// TIA Portal V17 export
// export: Created 2022-07-20T06:59:50.0989637Z, ExportSetting WithDefaults, DisplayName Totally Integrated Automation Portal, DisplayVersion V17, DisplayName TIA Portal Openness, DisplayVersion V17, DisplayName TIA Portal Version Control Interface, DisplayVersion V17, DisplayName SINAMICS Startdrive Advanced, DisplayVersion V17, DisplayName SINAMICS Startdrive G130, G150, S120, S150, SINAMICS MV, S210, DisplayVersion V17, DisplayName SINAMICS Startdrive G110M, G120, G120C, G120D, G120P, G115D, DisplayVersion V17, DisplayName STEP 7 Professional, DisplayVersion V17, DisplayName STEP 7 Safety, DisplayVersion V17, DisplayName WinCC Advanced, DisplayVersion V17
FUNCTION_BLOCK "FB10022_Average"   // FB10022, LAD
{ S7_Optimized_Access := 'TRUE' }
VERSION : 0.1
// stored: AutoNumber false, IsIECCheckEnabled false, IsRetainMemResEnabled false, MemoryReserve 100, SetENOAutomatically false, UDAEnableTagReadback false
   VAR_INPUT
      Value : Real;
      Clock : Bool;
      Clear : Bool;
   END_VAR
   VAR_OUTPUT
      Result : Real;
   END_VAR
   VAR_IN_OUT
      Items : Array[*] of Real;
   END_VAR
   VAR
      R_TRIG_Clock : R_TRIG;
      statItemNumber { S7_SetPoint := 'True'} : DInt;
      statStartElement : DInt;
      statEndElement : DInt;
      statItemsFull : Bool;
   END_VAR
   VAR_TEMP
      iItem : Int;
   END_VAR
BEGIN

REGION Network 1 (SCL): First Scan
   IF "FirstScan" THEN
       #statStartElement := LOWER_BOUND(ARR := #Items, DIM := 1);
       #statEndElement := UPPER_BOUND(ARR := #Items, DIM := 1);

       FOR #iItem := #statStartElement TO #statEndElement DO
           #Items[#iItem] := 0.0;
       END_FOR;

       #statItemNumber := #statStartElement;
       #statItemsFull := FALSE;

   END_IF;
END_REGION

REGION Network 2 (SCL): Edge Signals & Timers
   REGION EDGE SIGNALS
       #R_TRIG_Clock(CLK := #Clock);

   END_REGION

   REGION TIMERS
   END_REGION
END_REGION

REGION Network 3 (SCL): Add an item and get data average
   IF #R_TRIG_Clock.Q THEN

       #Items[#statItemNumber] := #Value;
       #statItemNumber := #statItemNumber + 1;

       IF #statItemNumber > #statEndElement THEN
           #statItemNumber := #statStartElement;
           #statItemsFull := TRUE;
       END_IF;

       #Result := 0.0;

       IF #statItemsFull THEN
           FOR #iItem := #statStartElement TO #statEndElement DO
               #Result := #Items[#iItem] + #Result;
           END_FOR;

           #Result := #Result / (#statEndElement - #statStartElement + 1);
       ELSE
           FOR #iItem := #statStartElement TO #statItemNumber DO
               #Result := #Items[#iItem] + #Result;
           END_FOR;

           #Result := #Result / (#statItemNumber - #statStartElement);
       END_IF;
   END_IF;
END_REGION

REGION Network 4 (SCL): Clear all data
   IF #Clear THEN
       FOR #iItem := #statStartElement TO #statEndElement DO
           #Items[#statItemNumber] := 0.0;
       END_FOR;

       #statItemNumber := #statStartElement;
       #statItemsFull := FALSE;
       #Result := 0.0;
   END_IF;
END_REGION
END_FUNCTION_BLOCK
